SYSTEM FillerUnit (* Unit Filler, generated from its unit specification *)
  (* Standard: 61499-2 *)
  APPLICATION Filler (* Unit Filler (generated by unitgen) *)
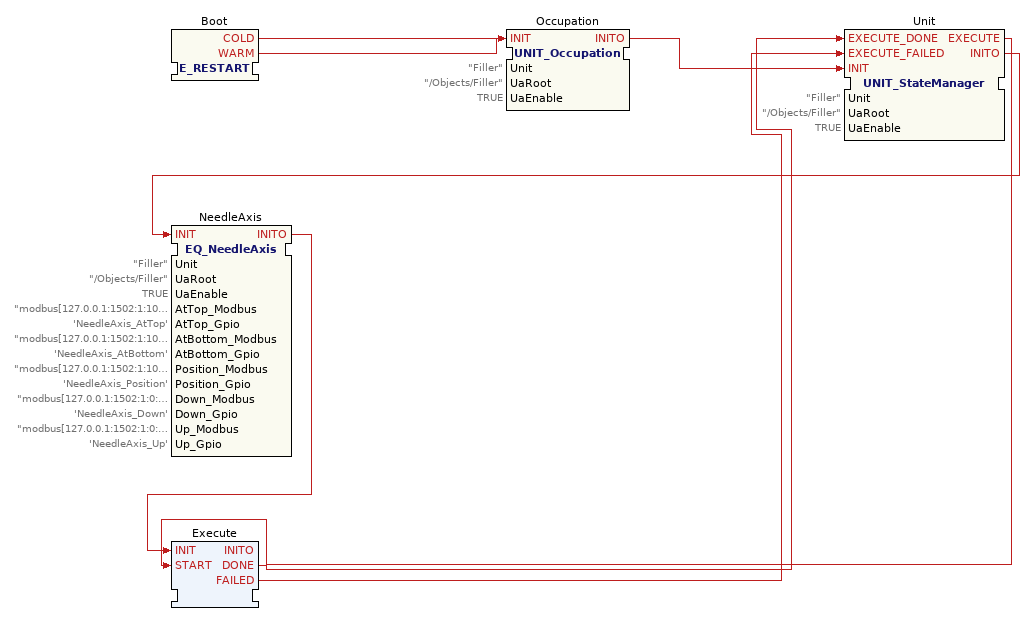
    FBS
      Boot : iec61499::events::E_RESTART;
      Occupation : unitlib::UNIT_Occupation(Unit := "Filler", UaRoot := "/Objects/Filler", UaEnable := TRUE);
      Unit : unitlib::UNIT_StateManager(Unit := "Filler", UaRoot := "/Objects/Filler", UaEnable := TRUE);
      NeedleAxis : filler::EQ_NeedleAxis(Unit := "Filler", UaRoot := "/Objects/Filler", UaEnable := TRUE, AtTop_Modbus := "modbus[127.0.0.1:1502:1:10:d0:]", AtTop_Gpio := 'NeedleAxis_AtTop', AtBottom_Modbus := "modbus[127.0.0.1:1502:1:10:d1:]", AtBottom_Gpio := 'NeedleAxis_AtBottom', Position_Modbus := "modbus[127.0.0.1:1502:1:10:i1:]", Position_Gpio := 'NeedleAxis_Position', Down_Modbus := "modbus[127.0.0.1:1502:1:0::c0]", Down_Gpio := 'NeedleAxis_Down', Up_Modbus := "modbus[127.0.0.1:1502:1:0::c2]", Up_Gpio := 'NeedleAxis_Up');
    END_FBS
    SUBAPPLICATION Execute (* PackML Execute procedure: skill instances chained SUCCESS -> START; any FAILURE fails the procedure *)
      EVENT_INPUT
        INIT : EInit;
        START;
      END_EVENT
      EVENT_OUTPUT
        INITO : EInit;
        DONE;
        FAILED;
      END_EVENT
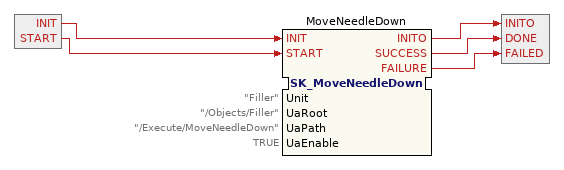
      FBS
        MoveNeedleDown : filler::SK_MoveNeedleDown(Unit := "Filler", UaRoot := "/Objects/Filler", UaPath := "/Execute/MoveNeedleDown", UaEnable := TRUE);
      END_FBS
      EVENT_CONNECTIONS
        INIT TO MoveNeedleDown.INIT;
        START TO MoveNeedleDown.START;
        MoveNeedleDown.INITO TO INITO;
        MoveNeedleDown.SUCCESS TO DONE;
        MoveNeedleDown.FAILURE TO FAILED;
      END_CONNECTIONS
    END_SUBAPPLICATION
    EVENT_CONNECTIONS
      Boot.COLD TO Occupation.INIT;
      Boot.WARM TO Occupation.INIT;
      Unit.EXECUTE TO Execute.START;
      Execute.DONE TO Unit.EXECUTE_DONE;
      Execute.FAILED TO Unit.EXECUTE_FAILED;
      Occupation.INITO TO Unit.INIT;
      Unit.INITO TO NeedleAxis.INIT;
      NeedleAxis.INITO TO Execute.INIT;
    END_CONNECTIONS
  END_APPLICATION
  DEVICE FORTE_PC : iec61499::system::FORTE_PC(MGR_ID := "localhost:61499")
    {SET_ATTRIBUTE(Profile, HOLOBLOC)} (* device profile *)
    RESOURCE RES : iec61499::system::EMB_RES
    END_RESOURCE
  END_DEVICE
  MAPPINGS
    Filler.Boot ON FORTE_PC.RES;
    Filler.Occupation ON FORTE_PC.RES;
    Filler.Unit ON FORTE_PC.RES;
    Filler.NeedleAxis ON FORTE_PC.RES;
    Filler.Execute ON FORTE_PC.RES;
  END_MAPPINGS
END_SYSTEM
